(* IEC 61131-3 sources: teller/JD_Teller_LC2_V11/Class/SetPassword, 1 file *)

(* ---- SetPassword.st ---- *)
(*!
<Class
	Name               = "SetPassword"
	Revision           = "0.0"
	RealtimeTask       = "false"
	CyclicTask         = "false"
	BackgroundTask     = "false"
	Sigmatek           = "false"
	OSInterface        = "false"
	HighPriority       = "false"
	Automatic          = "false"
	UpdateMode         = "Prescan"
	SharedCommandTable = "true"
	Objectsize         = "(284,120)">
	<Channels>
		<Server Name="ClassSvr" Visualized="false" Initialize="false" WriteProtected="true" Retentive="false"/>
		<Client Name="ActKey" Required="true" Internal="false"/>
		<Client Name="Always" Required="true" Internal="false"/>
		<Client Name="PreSetKey" Required="true" Internal="false"/>
	</Channels>
</Class>
*)
SetPassword : CLASS
  //Servers:
	ClassSvr 	: SvrChCmd_DINT;
  //Clients:
	Always 	: CltCh_DINT;
	ActKey 	: CltCh_DINT;
	PreSetKey 	: CltCh_DINT;
  //Variables:
  //Functions:

	FUNCTION VIRTUAL GLOBAL Init;
  //Tables:
	FUNCTION @STD
		VAR_OUTPUT
			ret_code	: CONFSTATES;
		END_VAR;
	FUNCTION GLOBAL TAB @CT_;
END_CLASS;

FUNCTION VIRTUAL GLOBAL SetPassword::Init

  if Always then
    ActKey := PreSetKey;
    ActKey.Write(input:=ActKey);
  else
    ActKey := ActKey.read();
    if ActKey = 0 then
      ActKey := PreSetKey;
      ActKey.Write(input:=ActKey);
    end_if;
  end_if;

END_FUNCTION
